# EPICS autosave request: iocBoot/gmca_23o_ioc1/dbSave/bluiceRun.req
$(P)runStatus
$(P)nextFrame
$(P)runLabel
$(P)fileroot
$(P)directory
$(P)startFrameLabel
$(P)axisMotor
$(P)startAngle
$(P)endAngle
$(P)delta
$(P)wedgeSize
$(P)exposureTime
$(P)distance
$(P)numEnergy
$(P)energy1
$(P)energy2
$(P)energy3
$(P)energy4
$(P)energy5
$(P)modeIndex
$(P)inverseOn
$(P)updated
